{attribute 'GeneratedUsingTerminal: EP2338-0001-0018'}
{attribute addProperty BoxType "EP2338-0001-0018"}
{attribute addProperty Description "EP2338-0001 8 Ch. Dig. Input/Output 24V, 0,5A, M8"}
{attribute addProperty Physics "YY"}
{attribute addProperty Id "Channel_1AT %I*Channel_830843C11Channel_2AT %I*Channel_830843C11Channel_3AT %I*Channel_830843C11Channel_4AT %I*Channel_830843C11Channel_5AT %I*Channel_830843C11Channel_6AT %I*Channel_830843C11Channel_7AT %I*Channel_830843C11Channel_8AT %I*Channel_830843C11Channel_9AT %Q*Channel_42CA91F71Channel_10AT %Q*Channel_42CA91F71Channel_11AT %Q*Channel_42CA91F71Channel_12AT %Q*Channel_42CA91F71Channel_13AT %Q*Channel_42CA91F71Channel_14AT %Q*Channel_42CA91F71Channel_15AT %Q*Channel_42CA91F71Channel_16AT %Q*Channel_42CA91F71WcStateAT %I*WcState_9091E0EB2InfoDataAT %I*InfoData_6F19DB2B2"}
{attribute addProperty CRC "1989786870"}
{attribute addProperty Size "20"}
TYPE EP2338_7699BCF6 EXTENDS EtcSlaveBoxBase_77A0E4A7 :
STRUCT
	{attribute addProperty Name "Channel_1"}
	Channel_1 : Channel_830843C1;
	{attribute addProperty Name "Channel_2"}
	Channel_2 : Channel_830843C1;
	{attribute addProperty Name "Channel_3"}
	Channel_3 : Channel_830843C1;
	{attribute addProperty Name "Channel_4"}
	Channel_4 : Channel_830843C1;
	{attribute addProperty Name "Channel_5"}
	Channel_5 : Channel_830843C1;
	{attribute addProperty Name "Channel_6"}
	Channel_6 : Channel_830843C1;
	{attribute addProperty Name "Channel_7"}
	Channel_7 : Channel_830843C1;
	{attribute addProperty Name "Channel_8"}
	Channel_8 : Channel_830843C1;
	{attribute addProperty Name "Channel_9"}
	Channel_9 : Channel_42CA91F7;
	{attribute addProperty Name "Channel_10"}
	Channel_10 : Channel_42CA91F7;
	{attribute addProperty Name "Channel_11"}
	Channel_11 : Channel_42CA91F7;
	{attribute addProperty Name "Channel_12"}
	Channel_12 : Channel_42CA91F7;
	{attribute addProperty Name "Channel_13"}
	Channel_13 : Channel_42CA91F7;
	{attribute addProperty Name "Channel_14"}
	Channel_14 : Channel_42CA91F7;
	{attribute addProperty Name "Channel_15"}
	Channel_15 : Channel_42CA91F7;
	{attribute addProperty Name "Channel_16"}
	Channel_16 : Channel_42CA91F7;
	{attribute addProperty Name "WcState"}
	WcState : WcState_9091E0EB;
	{attribute addProperty Name "InfoData"}
	InfoData : InfoData_6F19DB2B;
END_STRUCT
END_TYPE

(* stored: Version 1.2.0.0, ProductVersion 3.1.4024.9
   DUT EP2338_7699BCF6: Id {202d65f0-c897-4ace-9257-2e866c330143} *)
